(* PLC project Tc2_Utilities.ULARGE_TO_LARGE Demo, tc3-libraries-kb TwinCAT 3.1 *)
(* stored: creationDateTime 2026-05-12T12:00:00, modificationDateTime 2026-05-12T12:00:00 *)

PROGRAM P_Demo_ULARGE_TO_LARGE
  VAR
    uliRaw : T_ULARGE_INTEGER;
    liSigned : T_LARGE_INTEGER;
    bConvert : BOOL;
  END_VAR

            // ============================================================
// Tc2_Utilities.ULARGE_TO_LARGE 演示程序（FUNCTION，单周期触发）
// ============================================================
// 场景：无符号读回的位串希望按有符号显示（比如负温度的差值表示）。
// 价值：替代字段复制。
// 验证步骤：
//   1. 把本 PROGRAM 加到 PlcTask 调用列表
//   2. 编译 + 登录
//   3. 在线把 b... 触发位置 TRUE 一个周期
//   4. 观察输出变量是否符合期望
// ============================================================

IF bConvert THEN
    liSigned := ULARGE_TO_LARGE(uliRaw);
    bConvert := FALSE;
END_IF;

          
END_PROGRAM
